PROGRAM MAIN
VAR
	bohrmaschine: Bohrmaschine;
	stConfig: ST_Config;
	
	trigOnce: R_TRIG();
END_VAR



// TODO Input validation, error management
// TODO init functions, start-stop

// TODO via ADS
stConfig.rLaenge := 300;
stConfig.rBreite := 300;
stConfig.rDicke := 20.2;

trigOnce(CLK := TRUE);
IF trigOnce.Q THEN
	F_Log('Once');
	bohrmaschine.Config(stConfig);
	bohrmaschine.Start();
END_IF

bohrmaschine();

END_PROGRAM

(* stored: Version 1.1.0.1, ProductVersion 3.1.4024.3
   POU MAIN: Id {a92a02fc-7e74-4f5b-8c2e-324e945c69b3}, SpecialFunc None *)
